{attribute addProperty BoxType "EJ2914-0000-0017"}
{attribute addProperty Id "FSoE_CommandUSINT811FSOUT_Module_Channel_1_OutputBIT10.1251FSOUT_Module_Channel_2_OutputBIT10.1252FSOUT_Module_Channel_3_OutputBIT10.1253FSOUT_Module_Channel_4_OutputBIT10.1254FSOUT_Module_ErrAckBIT10.1251FSoE_CRC_000UINT1623FSoE_Connection_IDUINT1622"}
{attribute addProperty CRC "277349313"}
{attribute addProperty SizeInBites "48"}
{attribute addProperty SizeInBytes "6"}
TYPE FSOE_108803C1 :
STRUCT
	{attribute addProperty Name "FSoE_Command"}
	FSoE_Command : USINT;
	{attribute addProperty Name "FSOUT_Module_Channel_1_Output"}
	FSOUT_Module_Channel_1_Output : BOOL;
	{attribute addProperty Name "FSOUT_Module_Channel_2_Output"}
	FSOUT_Module_Channel_2_Output : BOOL;
	{attribute addProperty Name "FSOUT_Module_Channel_3_Output"}
	FSOUT_Module_Channel_3_Output : BOOL;
	{attribute addProperty Name "FSOUT_Module_Channel_4_Output"}
	FSOUT_Module_Channel_4_Output : BOOL;
	{attribute addProperty Name "FSOUT_Module_ErrAck"}
	FSOUT_Module_ErrAck : BOOL;
	{attribute 'hide'}
	reserve_1_BIT_0 : BOOL;
	{attribute 'hide'}
	reserve_1_BIT_1 : BOOL;
	{attribute 'hide'}
	reserve_1_BIT_2 : BOOL;
	{attribute addProperty Name "FSoE_CRC_000"}
	FSoE_CRC_000 : UINT;
	{attribute addProperty Name "FSoE_Connection_ID"}
	FSoE_Connection_ID : UINT;
END_STRUCT
END_TYPE

(* stored: Version 1.2.0.0, ProductVersion 3.1.4024.9
   DUT FSOE_108803C1: Id {92057828-449e-4f4f-af6f-2b480997936d} *)
